// TIA Portal V17 export
// export: Created 2022-02-03T14:45:18.2093983Z, ExportSetting WithDefaults, DisplayName Totally Integrated Automation Portal, DisplayVersion V17, DisplayName TIA Portal Openness, DisplayVersion V17, DisplayName TIA Portal Version Control Interface, DisplayVersion V17, DisplayName SINAMICS Startdrive Advanced, DisplayVersion V17, DisplayName SINAMICS Startdrive G130, G150, S120, S150, SINAMICS MV, S210, DisplayVersion V17, DisplayName SINAMICS Startdrive G110M, G120, G120C, G120D, G120P, G115D, DisplayVersion V17, DisplayName STEP 7 Professional, DisplayVersion V17, DisplayName STEP 7 Safety, DisplayVersion V17, DisplayName WinCC Advanced, DisplayVersion V17
ORGANIZATION_BLOCK "Startup"   // OB100, LAD, Startup
TITLE = "Complete Restart"
{ S7_Optimized_Access := 'TRUE' }
VERSION : 0.1
// stored: AutoNumber true, IsIECCheckEnabled false, SetENOAutomatically false
   VAR_INPUT
      LostRetentive : Bool;   // True if retentive data are lost
      LostRTC : Bool;   // True if date and time are lost
   END_VAR
   VAR_TEMP
      tempRET_VAL : Int;
      tempTOP_SI : SI_classic;
      tempSTARTUP_SI : SI_none;
   END_VAR
BEGIN

REGION Network 1
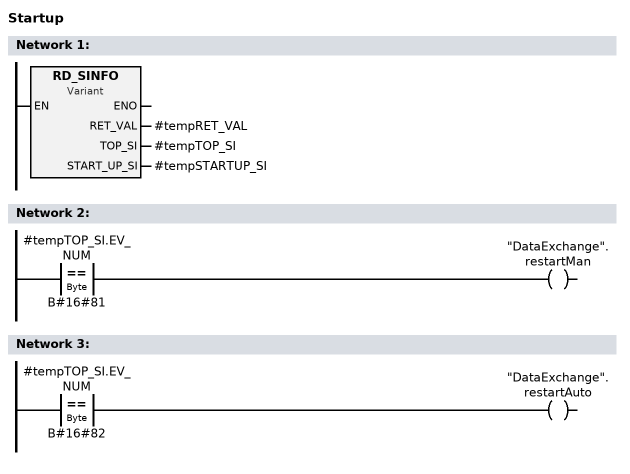
   RUNG wire#powerrail
      { S7_Templates := "si_type := Variant" } RD_SINFO(RET_VAL => #tempRET_VAL, TOP_SI => #tempTOP_SI, START_UP_SI => #tempSTARTUP_SI)
   END_RUNG
   // the same network as SCL:
   #tempRET_VAL := RD_SINFO(TOP_SI => #tempTOP_SI, START_UP_SI => #tempSTARTUP_SI);
END_REGION

REGION Network 2
   RUNG wire#powerrail
      { S7_Templates := "SrcType := Byte" } EQ_Contact(in1 := #tempTOP_SI.EV_NUM, in2 := B#16#81)
      Coil( "DataExchange".restartMan )
   END_RUNG
   // the same network as SCL:
   "DataExchange".restartMan := #tempTOP_SI.EV_NUM = B#16#81;
END_REGION

REGION Network 3
   RUNG wire#powerrail
      { S7_Templates := "SrcType := Byte" } EQ_Contact(in1 := #tempTOP_SI.EV_NUM, in2 := B#16#82)
      Coil( "DataExchange".restartAuto )
   END_RUNG
   // the same network as SCL:
   "DataExchange".restartAuto := #tempTOP_SI.EV_NUM = B#16#82;
END_REGION
END_ORGANIZATION_BLOCK
